FUNCTION_BLOCK FB_exitLoadTrigger
VAR_INPUT
	input_right : BOOL;
	input_left : BOOL;
	input_forward : BOOL;
	
END_VAR
VAR_OUTPUT
	leftExitEdge : BOOL;
	rightExitEdge: BOOL;
	forwardExitEdge : BOOL;
END_VAR
VAR
	f_trig_left : Tc2_Standard.F_TRIG;
	f_trig_right : Tc2_Standard.F_TRIG;
	f_trig_forward : Tc2_Standard.F_TRIG;
END_VAR

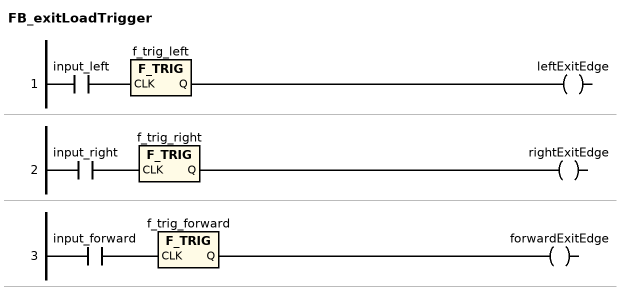
// NETWORK 1
f_trig_left(CLK := input_left); // F_TRIG
leftExitEdge := f_trig_left.Q;

// NETWORK 2
f_trig_right(CLK := input_right); // F_TRIG
rightExitEdge := f_trig_right.Q;

// NETWORK 3
f_trig_forward(CLK := input_forward); // F_TRIG
forwardExitEdge := f_trig_forward.Q;

END_FUNCTION_BLOCK

(* stored: Version 1.1.0.1, ProductVersion 3.1.4024.13
   POU FB_exitLoadTrigger: Id {e2d4fcfc-6065-40b6-9cb1-25e7234dd26e}, SpecialFunc None *)
